TYPE "Straightener_Manager"
VERSION : 0.1
// Block: Straightener_Manager
   STRUCT
      Feed : PositioningMachine_Manager;
      Lift_Entry : ValveMachine_Manager;
      Lift_Exit : ValveMachine_Manager;
   END_STRUCT;

END_TYPE
